# EPICS autosave request: ADApp/Db/NDOverlayN_settings.req
$(P)$(R)Name
$(P)$(R)Use
$(P)$(R)PositionXLink.DOL
$(P)$(R)PositionX
$(P)$(R)PositionYLink.DOL
$(P)$(R)PositionY
$(P)$(R)SizeXLink.DOL
$(P)$(R)SizeX
$(P)$(R)SizeYLink.DOL
$(P)$(R)SizeY
$(P)$(R)DrawMode
$(P)$(R)Shape
$(P)$(R)Red
$(P)$(R)Green
$(P)$(R)Blue
$(P)$(R)TimeStampFormat
$(P)$(R)Font
$(P)$(R)DisplayText
